TYPE T_Ctrl_SIf_MOD_Cfg :
STRUCT
	eTyp: E_Typ_MOD;
END_STRUCT
END_TYPE

(* stored: Version 1.1.0.1, ProductVersion 3.1.0.25
   DUT T_Ctrl_SIf_MOD_Cfg: Id {19ba0013-d082-4558-b8d4-6e162f54dbc3} *)
